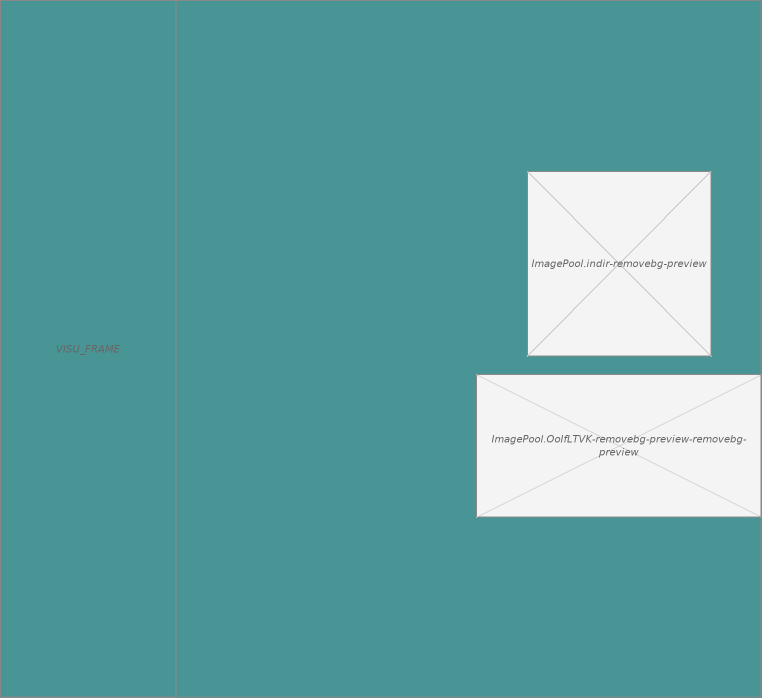
VISUALIZATION Visualization_3  // 762x698
    Image (527,171 184x185), image: ImagePool.indir-removebg-preview
    Image (476,374 286x143), image: ImagePool.OoIfLTVK-removebg-preview-removebg-preview
    Frame (0,0 176x698)
        shows VISU_FRAME(sDayTime := MAIN.DMY_LocalTime, sTime := MAIN.HMS_LocalTime)
END_VISUALIZATION

(* stored: Version 1.1.0.1, ProductVersion 3.1.4024.4
   Visu Visualization_3: Id {dcff6593-9745-4ace-821c-d7ba40215569} *)
